// TIA Portal V20 export
// export: Created 2025-12-01T14:57:05.0864165Z, ExportSetting None, DisplayName Totally Integrated Automation Portal, DisplayVersion V20 Update 3, DisplayName TIA Portal Openness, DisplayVersion V20 Update 3, DisplayName TIA Portal Version Control Interface, DisplayVersion V20 Update 3, DisplayName STEP 7 Professional, DisplayVersion V20 Update 3, DisplayName STEP 7 Safety, DisplayVersion V20 Update 2, DisplayName WinCC Basic/Comfort/Advanced, DisplayVersion V20 Update 3, DisplayName WinCC Professional, DisplayVersion V20 Update 3, DisplayName WinCC Unified, DisplayVersion V20 Update 3
FUNCTION "FC815_EventosEnv_Control" : Void   // FC815, LAD
{ S7_Optimized_Access := 'FALSE' }
AUTHOR : TRACKING
NAME : 20141014
VERSION : 4.0
// stored: AutoNumber false, SetENOAutomatically false
   VAR_INPUT
      NumJDT : UInt;
   END_VAR
   VAR_TEMP
      P_Eventos : DWord;
      DBEventos : Word;
      NumDBEventos : UInt;
      MaxBytes : UInt;
      NumBytes : UInt;
      InicioBucleMesas : UInt;
      FinalBulceMesas : UInt;
      MesaDeJDT02 : Bool;
      JDT02_Activo : Bool;
      NumMesa : UInt;
      NumeroUT : UInt;
      EventoInforme : UInt;
      Offset : UInt;
      Valor : UDInt;
      Evento : UDInt;
      Motivo : UDInt;
      ValorReturn : Int;
      Cero : Byte;
   END_VAR
BEGIN

NETWORK
TITLE = Inicializar
/////////////////////////////////////////////////////////////////////////////////////
/// Inicio --> Se esta en el  JDT02

      SET;
      R     #JDT02_Activo;

      L     "JDT1_NDB_EventosEmi";
      T     #DBEventos;
      T     #NumDBEventos;
      L     "JDT1_MaxBytes";
      T     #MaxBytes;

      L     "JDT1_InicioBucleMesas";  // Tamaño Bucles
      T     #InicioBucleMesas;
      L     "JDT1_FinalBucleMesas";
      T     #FinalBulceMesas;


      L     #NumJDT;
      L     2;
      <>I;
      JC    NoJDT02;

      SET;
      S     #JDT02_Activo;

      L     "JDT2_NDB_EventosEmi";
      T     #DBEventos;
      T     #NumDBEventos;
      L     "JDT2_MaxBytes";
      T     #MaxBytes;

      L     "JDT2_InicioBucleMesas";  // Tamaño Bucles
      T     #InicioBucleMesas;
      L     "JDT2_FinalBucleMesas";
      T     #FinalBulceMesas;

NoJDT02:NOP   0;

/// Inicio --> Se esta en el JDT 02
/////////////////////////////////////////////////////////////////////////////////////



NETWORK
TITLE = Generar Eventos de las UT's
// - Recorrer todas las Mesas Buscando UT'que necesiten generar Eventos
//   Dos bucles anidados Mesas y UT's dentro de las Mesas ( No se hace)
// - Recorrer todas las UT's (Se hace
/////////////////////////////////////////////////////////////////////////////////////
// --- Recorrer todas las Mesas

      L     #InicioBucleMesas;
      T     #NumMesa;

Inicio_BucleDeMesas:NOP   0;
///////////////////////////////////////////////////////////////////////////////////////
/// Mirar si esta defincido como mesa de tracking

      SET;
      AN    "DB850_DefinicionMesas".Mesa[#NumMesa].ConfigMesa.MesaPaso;
      AN    "DB850_DefinicionMesas".Mesa[#NumMesa].ConfigMesa.MesaCruce;
      AN    "DB850_DefinicionMesas".Mesa[#NumMesa].ConfigMesa.MesaMultiplesDestinos;
      JC    Siguiente_BucleDeMesas;


///////////////////////////////////////////////////////////////////////////////////////
/// Mirar Si pertenece al JDT

      SET;
      X     "DB850_DefinicionMesas".Mesa[#NumMesa].ConfigMesa.MesaDeJDT02;
      XN    #JDT02_Activo;  // JDT01 o JDT02 ?
      =     #MesaDeJDT02;

      SET;
      AN    #MesaDeJDT02;
      JC    Siguiente_BucleDeMesas;


/////////////////////////////////////////////////////////////////////////////////////
/// Mirar Si Existe una UT en la Mesa

      L     "DB810_ColasMesas".Colas[#NumMesa].UT_PrimeraMesa;
      T     #NumeroUT;

      L     #NumeroUT;
      L     0;
      ==I;
      JC    Siguiente_BucleDeMesas;  // No hay UT's en la Mesa


///////////////////////////////////////////////////////////////////////////////////////
// --- Recorrer todas las UT's de la Mesa

Inicio_BucelDeUTs_DeMesa:NOP   0;

///////////////////////////////////////////////////////////////////////////////////////
// --- Comprobar Si hay que Enviar Eventos

// --- Informacion poor Cambio de Mesa de la UT
      SET;
      A     "DB812_UTs_Control".UT[#NumeroUT].EventosInformarJdT.CambiadaDeMesa;
      JC    EnviarEvento_CambiadaDeMesa;
      SET;
      A     "DB812_UTs_Control".UT[#NumeroUT].EventosInformarJdT.CambiadaPosicionUp;
      JC    EnviarEvento_CambiadaPosicionUp;
      SET;
      A     "DB812_UTs_Control".UT[#NumeroUT].EventosInformarJdT.CambiadaPosicionDown;
      JC    EnviarEvento_CambiadaPosicionDown;
      SET;
      A     "DB812_UTs_Control".UT[#NumeroUT].EventosInformarJdT.NoCambidaDeMesa;
      JC    EnviarEvento_MoCambiadaDeMesa;

// --- Informacion por la Duplicidad del Mckey por el Evento CREA
      SET;
      A     "DB812_UTs_Control".UT[#NumeroUT].EventosInformarJdT.DuplicidadMckey;
      JC    EnviarEvento_Duplicidad_UT;

// --- 2023 01 05 - Nuevo Sistema para Informar sobre la UT - Evento ?UT?
      SET;
      A     "DB812_UTs_Control".UT[#NumeroUT].EventosInformarJdT.PeticionDeDatos;
      JC    EnviarEvento_PeticionDeDatos;

// --- 2023 01 05 - Nuevo Sistema para Informar sobre la UT - Evento CHEQ
      SET;
      A     "DB812_UTs_Control".UT[#NumeroUT].EventosInformarJdT.ChequeoDelReset;
      JC    EnviarEvento_ChequeoDelReset;


// --- No Hay que Enviar Eventos
///////////////////////////////////////////////////////////////////////////////////////
///////////////////////////////////////////////////////////////////////////////////////

Siguiente_BucleDeUTs:NOP   0;

      L     "DB812_UTs_Control".UT[#NumeroUT].UT_SiguienteMesa;
      T     #NumeroUT;

      L     #NumeroUT;
      L     0;
      ==I;
      JC    Siguiente_BucleDeMesas;  // No hay mas UT's en la Mesa

      JU    Inicio_BucelDeUTs_DeMesa;  // Seguir recorriendo la Mesa


///////////////////////////////////////////////////////////////////////////////////////
// --- Continuar recorriendo el resto de Mesas

Siguiente_BucleDeMesas:NOP   0;
      L     #NumMesa;
      L     #FinalBulceMesas;
      >=I;
      JC    FinalFuncion;  // Ya no hay más UT's ?

      L     #NumMesa;  // +1, Para la Siguiente UT
      L     1;
      +I;
      T     #NumMesa;

      JU    Inicio_BucleDeMesas;  // Ir a mirar la siguiente UT



NETWORK
TITLE = Acciones
///////////////////////////////////////////////////////////////////////////////////////
EnviarEvento_CambiadaDeMesa:NOP   0;
      L     'CAMB';
      T     #Motivo;
      L     'MOV!';
      T     #Evento;
      JU    EmitirEvento;  // Evento - MOV! - CAMBIO


///////////////////////////////////////////////////////////////////////////////////////
EnviarEvento_MoCambiadaDeMesa:NOP   0;
      L     'NCAM';
      T     #Motivo;
      L     'MOV!';
      T     #Evento;
      JU    EmitirEvento;  // Evento - MOV! - NoCAMBIO


///////////////////////////////////////////////////////////////////////////////////////
EnviarEvento_CambiadaPosicionDown:NOP   0;
      L     'CAMD';
      T     #Motivo;
      L     'INFO';
      T     #Evento;
      JU    EmitirEvento;  // Evento - INFO - CAMBIO DOWN


///////////////////////////////////////////////////////////////////////////////////////
EnviarEvento_CambiadaPosicionUp:NOP   0;
      L     'CAMU';
      T     #Motivo;
      L     'INFO';
      T     #Evento;
      JU    EmitirEvento;  // Evento - INFO - CAMBIO UP


///////////////////////////////////////////////////////////////////////////////////////
EnviarEvento_Duplicidad_UT:NOP   0;
      L     'DUPL';
      T     #Motivo;
      L     'INFO';
      T     #Evento;
      JU    EmitirEvento;  // Evento - INFO - DUPLICIDAD DE MCKEY



NETWORK
TITLE = Evento de Estado de Inicio de Bucle
EmitirEvento:NOP   0;

///////////////////////////////////////////////////////////////////////////////////////
// ---   Formateo del Evento de Estado del Dispositivo
// ---   * Mirar si hay sitio para generar el nuevo evento
// ---       * Inicializo NumBytes y Puntero al DB de Eventos Generados
// ---       * Calcula el tamaño de bytes que hay en el DB de Eventos Generados
// ---       * Comprobar si hay sitio para un evento más
// ---   *  Formatear el evento de Estado de Inicio de Bucle  INI!
///////////////////////////////////////////////////////////////////////////////////////


///////////////////////////////////////////////////////////////////////////////////////
// --- Mirar si hay sitio para generar un evento más

      L     0;
      T     #NumBytes;  // Inicializo el numero de Bytes
      T     #P_Eventos;  // Inicializo el puntero de Eventos Generados

Inicio_BusquedaFinalEventos:NOP   0;
      OPN   DB [#DBEventos];  // Calcula el tamaño de bytes que hay en el DB
      L     DBB [#P_Eventos];
      L     0;
      ==I;
      JC    Fin_BusquedaFinalEventos;  // Buscamos el final del DB = 0

      OPN   DB [#DBEventos];
      L     DBB [#P_Eventos];
      L     ' ';
      ==I;
      JC    Fin_BusquedaFinalEventos;  // Buscamos el final del DB = ' '

      L     #P_Eventos;  // Incremento de P#1.0
      L     P#1.0;
      +D;
      T     #P_Eventos;

      JU    Inicio_BusquedaFinalEventos;  // Continuar con el siguiente posicion

Fin_BusquedaFinalEventos:NOP   0;
      L     #P_Eventos;  // Sacamos el NumBytes Escritos
      SRD   3;
      T     #NumBytes;

      L     #NumBytes;  // Miramos si hay sitio
      L     #MaxBytes;  // Max. que se pueden emitir, parametro
      >I;
      JC    FinalFuncion;  // No se pueden generar más eventos



///////////////////////////////////////////////////////////////////////////////////////
// --- Formatear el evento

      L     #P_Eventos;
      LAR2;  // Puntero al DB de Eventos Generados

      TAR2;  // Mirar si es el primer evento de la lista
      L     0;
      ==I;
      JC    NoEsInicio_ListaDeEventos;  // Es el primero

      OPN   DB [#DBEventos];
      L     ',';  // Separador entre eventos ','
      T     DBB [AR2, P#0.0];
      +AR2  P#1.0;

NoEsInicio_ListaDeEventos:NOP   0;

///////////////////////////////////////////////////////////////////////////////
// --- Cuerpo del Evento

      OPN   DB [#DBEventos];  // DB de Eventos Generados (A Emitir)
      L     '{';  // Inicio de Evento '{'
      T     DBB [AR2, P#0.0];
      +AR2  P#1.0;

      L     #Evento;  // --- Evento
      T     DBD [AR2, P#0.0];
      +AR2  P#4.0;


///////////////////////////////////////////////////////////////////////////////
      L     '[';  // Evento - Atributo Mckey '[MCKY]'
      T     DBB [AR2, P#0.0];
      L     'MCKY';
      T     DBD [AR2, P#1.0];
      L     ']';  // Evento - Atributo Mckey '[MCKY]'
      T     DBB [AR2, P#5.0];
      +AR2  P#6.0;

      L     "DB812_UTs_Control".UT[#NumeroUT].Mckey;
      T     #Valor;

// --- Convertir Valor a ASCII - Mckey
      TAR2;
      SRD   3;
      T     #NumBytes;  // Miro que offset tiene la String

      CALL  "FC893_Obtener_StringDelAtributo"
      ( DB_String := #NumDBEventos,
        OffsetIni := #NumBytes,
        Valor     := #Valor,
        OffsetFin := #Offset
      );  // Llamo a ObtenerStrinAtributo

      L     #Offset;
      SLD   3;
      LAR2;  // Recupero que offset tiene la String

// --- Ya esta convertido el Valor a ASCI - Fin Mckey


///////////////////////////////////////////////////////////////////////////////
      OPN   DB [#DBEventos];
      L     '[';  // Evento - Atributo Mesa Actual '[MESA]'
      T     DBB [AR2, P#0.0];
      L     'MESA';
      T     DBD [AR2, P#1.0];
      L     ']';
      T     DBB [AR2, P#5.0];
      +AR2  P#6.0;

      L     "DB812_UTs_Control".UT[#NumeroUT].MesaActual;
      T     #Valor;

// --- Convertir Valor a ASCII -  Mesa Actual
      TAR2;
      SRD   3;
      T     #NumBytes;  // Miro que offset tiene la String

      CALL  "FC893_Obtener_StringDelAtributo"
      ( DB_String := #NumDBEventos,
        OffsetIni := #NumBytes,
        Valor     := #Valor,
        OffsetFin := #Offset
      );  // Llamo a ObtenerStrinAtributo

      L     #Offset;
      SLD   3;
      LAR2;  // Recupero que offset tiene la String

// --- Ya esta convertido el Valor a ASCI - Fin Mesa Actual


///////////////////////////////////////////////////////////////////////////////
      OPN   DB [#DBEventos];
      L     '[';  // Evento - Atributo Mesa Actual '[MOTI]'
      T     DBB [AR2, P#0.0];
      L     'MOTI';
      T     DBD [AR2, P#1.0];
      L     ']';
      T     DBB [AR2, P#5.0];
      +AR2  P#6.0;

      L     #Motivo;
      T     DBD [AR2, P#0.0];
      +AR2  P#4.0;


///////////////////////////////////////////////////////////////////////////////
// --- Final del Evento

      OPN   DB [#DBEventos];  // DB de Eventos Generados (A Emitir)
      L     '}';  // --- Fin de Evento '}'
      T     DBB [AR2, P#0.0];
      +AR2  P#1.0;


///////////////////////////////////////////////////////////////////////////////
/// -- Dar  por enviado el evento

      SET;
      R     "DB812_UTs_Control".UT[#NumeroUT].EventosInformarJdT.CambiadaDeMesa;
      R     "DB812_UTs_Control".UT[#NumeroUT].EventosInformarJdT.CambiadaPosicionUp;
      R     "DB812_UTs_Control".UT[#NumeroUT].EventosInformarJdT.CambiadaPosicionDown;
      R     "DB812_UTs_Control".UT[#NumeroUT].EventosInformarJdT.NoCambidaDeMesa;
      R     "DB812_UTs_Control".UT[#NumeroUT].EventosInformarJdT.DuplicidadMckey;

      JU    Siguiente_BucleDeUTs;  //Final del Formateo del Elento



NETWORK
TITLE = Evento de Peticion de Datos de la UT >>> Evento ?UT?
///////////////////////////////////////////////////////////////////////////////
///////////////////////////////////////////////////////////////////////////////
///////////////////////////////////////////////////////////////////////////////
EnviarEvento_PeticionDeDatos:NOP   0;
      SET;  // --- Se puede ?
      L     "DB812_UTs_Control".UT[#NumeroUT].EstadoEventoAGenerar;
      L     0;  // EstaodEventoAGenerar = 0
      <>I;
      JC    Siguiente_BucleDeUTs;


///////////////////////////////////////////////////////////////////////////////
///////////////////////////////////////////////////////////////////////////////
///////////////////////////////////////////////////////////////////////////////
/// -- Dar por Activado el Evento DATO >>> Resepuesta por el Evento ?UT?
      L     110;  // 110 - Generar Evento de Refresco de Datos
      T     "DB812_UTs_Control".UT[#NumeroUT].EstadoEventoAGenerar;

      SET;
      R     "DB812_UTs_Control".UT[#NumeroUT].EventosInformarJdT.PeticionDeDatos;

      JU    Siguiente_BucleDeUTs;



NETWORK
TITLE = Evento de Chequeo de la UT >>> Evento CHEQ
EnviarEvento_ChequeoDelReset:NOP   0;
      SET;  // --- Se puede ?
      L     "DB812_UTs_Control".UT[#NumeroUT].EstadoEventoAGenerar;
      L     0;  // EstaodEventoAGenerar = 0
      <>I;
      JC    Siguiente_BucleDeUTs;


///////////////////////////////////////////////////////////////////////////////
///////////////////////////////////////////////////////////////////////////////
///////////////////////////////////////////////////////////////////////////////
/// -- Dar por Activado el Evento CHEQ! >>> Resepuesta por el Evento CHEQ
      L     145;  // 141 - Generar Evento de Chequeo del Reset
      T     "DB812_UTs_Control".UT[#NumeroUT].EstadoEventoAGenerar;

      SET;
      R     "DB812_UTs_Control".UT[#NumeroUT].EventosInformarJdT.ChequeoDelReset;

      JU    Siguiente_BucleDeUTs;



NETWORK
TITLE = Final de la Función
/////////////////////////////////////////////////////////////////////////////////////
FinalFuncion:NOP   0;


END_FUNCTION
